PROGRAM Output_Mapping
VAR
END_VAR

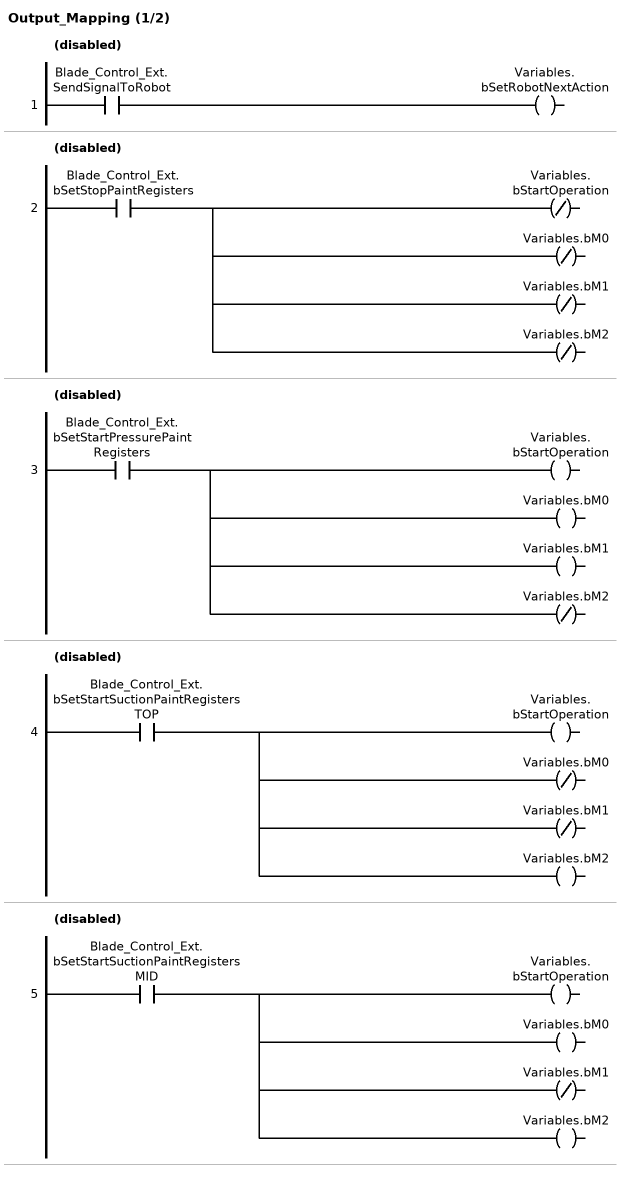
// NETWORK 1 (disabled)
// Variables.bSetRobotNextAction := Blade_Control_Ext.SendSignalToRobot;

// NETWORK 2 (disabled)
// Variables.bStartOperation := NOT Blade_Control_Ext.bSetStopPaintRegisters;
// Variables.bM0 := NOT Blade_Control_Ext.bSetStopPaintRegisters;
// Variables.bM1 := NOT Blade_Control_Ext.bSetStopPaintRegisters;
// Variables.bM2 := NOT Blade_Control_Ext.bSetStopPaintRegisters;

// NETWORK 3 (disabled)
// Variables.bStartOperation := Blade_Control_Ext.bSetStartPressurePaintRegisters;
// Variables.bM0 := Blade_Control_Ext.bSetStartPressurePaintRegisters;
// Variables.bM1 := Blade_Control_Ext.bSetStartPressurePaintRegisters;
// Variables.bM2 := NOT Blade_Control_Ext.bSetStartPressurePaintRegisters;

// NETWORK 4 (disabled)
// Variables.bStartOperation := Blade_Control_Ext.bSetStartSuctionPaintRegistersTOP;
// Variables.bM0 := NOT Blade_Control_Ext.bSetStartSuctionPaintRegistersTOP;
// Variables.bM1 := NOT Blade_Control_Ext.bSetStartSuctionPaintRegistersTOP;
// Variables.bM2 := Blade_Control_Ext.bSetStartSuctionPaintRegistersTOP;

// NETWORK 5 (disabled)
// Variables.bStartOperation := Blade_Control_Ext.bSetStartSuctionPaintRegistersMID;
// Variables.bM0 := Blade_Control_Ext.bSetStartSuctionPaintRegistersMID;
// Variables.bM1 := NOT Blade_Control_Ext.bSetStartSuctionPaintRegistersMID;
// Variables.bM2 := Blade_Control_Ext.bSetStartSuctionPaintRegistersMID;

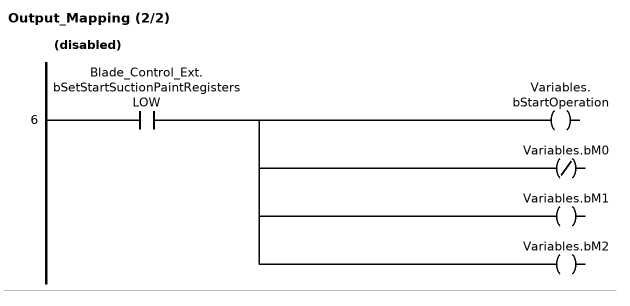
// NETWORK 6 (disabled)
// Variables.bStartOperation := Blade_Control_Ext.bSetStartSuctionPaintRegistersLOW;
// Variables.bM0 := NOT Blade_Control_Ext.bSetStartSuctionPaintRegistersLOW;
// Variables.bM1 := Blade_Control_Ext.bSetStartSuctionPaintRegistersLOW;
// Variables.bM2 := Blade_Control_Ext.bSetStartSuctionPaintRegistersLOW;

END_PROGRAM

(* stored: Version 1.1.0.1, ProductVersion 3.1.4020.6
   POU Output_Mapping: Id {4de51c9c-ccf7-4489-996a-1edbb2ffc9bf}, SpecialFunc None *)
